INTERFACE ITF_BaseHMIControlElement_Command

END_INTERFACE

(* stored: Version 1.1.0.1
   Itf ITF_BaseHMIControlElement_Command: Id {a455c728-d259-0a2b-0867-e5c3b1e949b9} *)
